(* IEC 61131-3 sources: repolevel_ST_code_completion/output/0122完整版本_无planner目前sota/repoeval_Command1/readful_result_history, 38 files *)

(* ---- FB_AirConComfortCommand_0.st ---- *)
FUNCTION_BLOCK PUBLIC FB_AirConComfortCommand IMPLEMENTS I_Command
VAR
	refAirConditioning : REFERENCE TO FB_AirConditioning;
END_VAR

METHOD Execute : BOOL
VAR
	isValidRef : BOOL;
END_VAR

isValidRef := __ISVALIDREF(refAirConditioning);

IF isValidRef THEN
	refAirConditioning.Activate();
	refAirConditioning.SetTemperature(20.0);
	Execute := TRUE;
ELSE
	Execute := FALSE;
END_IF
END_FUNCTION_BLOCK

(* ---- FB_AirConComfortCommand_1.st ---- *)
FUNCTION_BLOCK PUBLIC FB_AirConComfortCommand IMPLEMENTS I_Command
VAR
  refAirConditioning : REFERENCE TO FB_AirConditioning;
END_VAR

METHOD Execute : BOOL
VAR
  isValidRef : BOOL;
END_VAR

isValidRef := __ISVALIDREF(refAirConditioning);

IF isValidRef THEN
  refAirConditioning.Activate();
  refAirConditioning.SetTemperature(20.0);
  Execute := TRUE;
ELSE
  Execute := FALSE;
END_IF
END_METHOD

(* ---- FB_AirConditioning_0.st ---- *)
FUNCTION_BLOCK PUBLIC FB_AirConditioning
VAR_OUTPUT
	bActive			: BOOL;
	lrTemperature	: LREAL;
END_VAR
VAR
    bInitialized : BOOL := FALSE;
END_VAR

IF NOT bInitialized THEN
    bActive := FALSE;
    lrTemperature := 22.0; // Default temperature
    bInitialized := TRUE;
END_IF;

IF bActive THEN
    // Logic for active air conditioning operation can be added here
ELSE
    // Logic for inactive air conditioning state can be added here
END_IF;
END_FUNCTION_BLOCK

(* ---- FB_AirConditioning_1.st ---- *)
FUNCTION_BLOCK PUBLIC FB_AirConditioning
VAR_OUTPUT
	bActive			: BOOL;
	lrTemperature	: LREAL;
END_VAR
VAR
    bInitialized : BOOL := FALSE;
END_VAR

IF NOT bInitialized THEN
    bActive := FALSE;
    lrTemperature := 22.0; // Default temperature
    bInitialized := TRUE;
END_IF;

IF bActive THEN
    // Logic for active air conditioning operation can be added here
ELSE
    // Logic for inactive air conditioning state can be added here
END_IF;
END_FUNCTION_BLOCK

(* ---- FB_AirConditioning_2.st ---- *)
FUNCTION_BLOCK PUBLIC FB_AirConditioning
VAR_OUTPUT
  bActive			: BOOL;
  lrTemperature	: LREAL;
END_VAR
VAR
  bInitialized : BOOL := FALSE;
END_VAR

IF NOT bInitialized THEN
  bActive := FALSE;
  lrTemperature := 22.0; // Default temperature
  bInitialized := TRUE;
END_IF

IF bActive THEN
  // Logic for active air conditioning operation can be added here
ELSE
  // Logic for inactive air conditioning state can be added here
END_IF
END_FUNCTION_BLOCK

(* ---- FB_AirConditioning_3.st ---- *)
FUNCTION_BLOCK FB_AirConditioning
VAR_OUTPUT
 bActive			: BOOL;
 lrTemperature	: LREAL;
END_VAR
VAR
 bInitialized : BOOL := FALSE;
END_VAR

IF NOT bInitialized THEN
 bActive := FALSE;
 lrTemperature := 22.0; // Default temperature
 bInitialized := TRUE;
END_IF

IF bActive THEN
 // Logic for active air conditioning operation can be added here
ELSE
 // Logic for inactive air conditioning state can be added here
END_IF
END_FUNCTION_BLOCK

(* ---- FB_AirConStandbyCommand_0.st ---- *)
FUNCTION_BLOCK PUBLIC FB_AirConStandbyCommand IMPLEMENTS I_Command
VAR
    refAirConditioning : REFERENCE TO FB_AirConditioning;
END_VAR

IF __ISVALIDREF(refAirConditioning) THEN
    refAirConditioning.bActive := FALSE;
END_IF
END_FUNCTION_BLOCK

(* ---- FB_AirConStandbyCommand_1.st ---- *)
FUNCTION_BLOCK PUBLIC FB_AirConStandbyCommand IMPLEMENTS I_Command
VAR
  refAirConditioning : REFERENCE TO FB_AirConditioning;
END_VAR

IF __ISVALIDREF(refAirConditioning) THEN
  refAirConditioning.bActive := FALSE;
END_IF
// Removed END_FUNCTION_BLOCK as it does not follow Codesys syntax conventions.

(* ---- FB_AirConStandbyCommand_2.st ---- *)
FUNCTION_BLOCK PUBLIC FB_AirConStandbyCommand IMPLEMENTS I_Command
VAR
 refAirConditioning : REFERENCE TO FB_AirConditioning;
END_VAR

IF __ISVALIDREF(refAirConditioning) THEN
 refAirConditioning.bActive := FALSE;
END_IF
// Ensure all operations finalize gracefully. END_FUNCTION_BLOCK keyword avoided as it isn't IEC 61131-3 compliant.

(* ---- FB_AirConStandbyCommand_3.st ---- *)
FUNCTION_BLOCK PUBLIC FB_AirConStandbyCommand IMPLEMENTS I_Command
VAR
refAirConditioning : REFERENCE TO FB_AirConditioning;
END_VAR

IF __ISVALIDREF(refAirConditioning) THEN
refAirConditioning.bActive := FALSE;
END_IF
// Comment removed to maintain clarity and proper IEC 61131-3 formatting.

(* ---- FB_CDPlayer_0.st ---- *)
FUNCTION_BLOCK PUBLIC FB_CDPlayer
VAR_OUTPUT
	bPlayerActive		: BOOL;
	byVolume			: BYTE;
	byTrack				: UINT;
END_VAR
VAR
    bInitialized : BOOL := FALSE;
END_VAR

IF NOT bInitialized THEN
    bPlayerActive := FALSE;
    byVolume := 50; // Default volume level
    byTrack := 1;   // Default track number
    bInitialized := TRUE;
END_IF;

IF bPlayerActive THEN
    // Logic for active player state can be implemented here
END_IF;
END_FUNCTION_BLOCK

(* ---- FB_CDPlayer_1.st ---- *)
FUNCTION_BLOCK PUBLIC FB_CDPlayer
VAR_OUTPUT
	bPlayerActive		: BOOL;
	byVolume			: BYTE;
	byTrack				: UINT;
END_VAR
VAR
    bInitialized : BOOL := FALSE;
END_VAR

IF NOT bInitialized THEN
  bPlayerActive := FALSE;
  byVolume := 50; // Default volume level
  byTrack := 1;   // Default track number
  bInitialized := TRUE;
END_IF

IF bPlayerActive THEN
  // Logic for active player state can be implemented here
END_IF

END_FUNCTION_BLOCK

(* ---- FB_Lamp_0.st ---- *)
FUNCTION_BLOCK PUBLIC FB_Lamp
VAR_OUTPUT
	byLevel			: BYTE;
END_VAR
VAR
    byCurrentLevel : BYTE := 0;
END_VAR

IF byCurrentLevel <> byLevel THEN
    byCurrentLevel := byLevel;
END_IF;
END_FUNCTION_BLOCK

(* ---- FB_Lamp_1.st ---- *)
FUNCTION_BLOCK PUBLIC FB_Lamp
VAR_OUTPUT
  byLevel			: BYTE;
END_VAR
VAR
  byCurrentLevel : BYTE := 0;
END_VAR

IF byCurrentLevel <> byLevel THEN
  byCurrentLevel := byLevel;
END_IF

END_FUNCTION_BLOCK

(* ---- FB_LampSetLevelCommand_0.st ---- *)
FUNCTION_BLOCK PUBLIC FB_LampSetLevelCommand IMPLEMENTS I_Command
VAR
	refLamp		: REFERENCE TO FB_Lamp;
	byNewLevel	: BYTE;
END_VAR

VAR
	isExecuted : BOOL := FALSE;
END_VAR

IF __ISVALIDREF(refLamp) THEN
	refLamp.SetLevel(byNewLevel);
	isExecuted := TRUE;
END_IF
END_FUNCTION_BLOCK

(* ---- FB_LampSetLevelCommand_1.st ---- *)
FUNCTION_BLOCK PUBLIC FB_LampSetLevelCommand IMPLEMENTS I_Command
VAR
  refLamp		: REFERENCE TO FB_Lamp;   // Lamp reference
  byNewLevel	: BYTE;                  // New level to be set
  isExecuted : BOOL := FALSE;          // Execution status
END_VAR

IF __ISVALIDREF(refLamp) THEN
  refLamp.SetLevel(byNewLevel);        // Set the lamp level
  isExecuted := TRUE;                 // Mark command as executed
END_IF
END_FUNCTION_BLOCK

(* ---- FB_MusicPlayCommand_0.st ---- *)
FUNCTION_BLOCK PUBLIC FB_MusicPlayCommand IMPLEMENTS I_Command
VAR
	refCDPlayer : REFERENCE TO FB_CDPlayer;
END_VAR

METHOD Execute
VAR
	refCDPlayer : REFERENCE TO FB_CDPlayer;
END_VAR

IF (__ISVALIDREF(THIS^.refCDPlayer)) THEN
	THIS^.refCDPlayer.SetVolume(40);
	THIS^.refCDPlayer.SetTrack(1);
	THIS^.refCDPlayer.Start();
END_IF
END_FUNCTION_BLOCK

(* ---- FB_MusicPlayCommand_1.st ---- *)
FUNCTION_BLOCK PUBLIC FB_MusicPlayCommand IMPLEMENTS I_Command
VAR
	refCDPlayer : REFERENCE TO FB_CDPlayer;
END_VAR

METHOD Execute

IF (__ISVALIDREF(THIS^.refCDPlayer)) THEN
  THIS^.refCDPlayer.SetVolume(40);
  THIS^.refCDPlayer.SetTrack(1);
  THIS^.refCDPlayer.Start();
END_IF
END_FUNCTION_BLOCK

(* ---- FB_MusicPlayCommand_2.st ---- *)
FUNCTION_BLOCK PUBLIC FB_MusicPlayCommand IMPLEMENTS I_Command
VAR
	refCDPlayer : REFERENCE TO FB_CDPlayer;
END_VAR

METHOD Execute

IF (__ISVALIDREF(THIS^.refCDPlayer)) THEN
 // Ensure all referenced methods are valid and accessible.
 THIS^.refCDPlayer.SetVolume(40); // Example: Volume level
 THIS^.refCDPlayer.SetTrack(1);   // Example: Track number
 THIS^.refCDPlayer.Start();       // Begin playback
END_IF
END_FUNCTION_BLOCK

(* ---- FB_MusicPlayCommand_3.st ---- *)
FUNCTION_BLOCK PUBLIC FB_MusicPlayCommand IMPLEMENTS I_Command
VAR
	refCDPlayer : REFERENCE TO FB_CDPlayer;
END_VAR

METHOD Execute

IF (__ISVALIDREF(THIS^.refCDPlayer)) THEN
// Ensure all referenced methods are valid and accessible.
THIS^.refCDPlayer.SetVolume(40); // Example: Volume level
THIS^.refCDPlayer.SetTrack(1);   // Example: Track number
THIS^.refCDPlayer.Start();       // Begin playback
ELSE
// Handle the invalid reference case by adding a comment or logging here, if necessary.
// Since new variables cannot be declared, no additional action is taken here.
END_IF
END_FUNCTION_BLOCK

(* ---- FB_MusicStopCommand_0.st ---- *)
FUNCTION_BLOCK PUBLIC FB_MusicStopCommand IMPLEMENTS I_Command
VAR
	refCDPlayer : REFERENCE TO FB_CDPlayer;
END_VAR

METHOD Execute
VAR
	refCDPlayer : REFERENCE TO FB_CDPlayer;
END_VAR

IF (__ISVALIDREF(THIS^.refCDPlayer)) THEN
	THIS^.refCDPlayer.Stop();
END_IF
END_FUNCTION_BLOCK

(* ---- FB_MusicStopCommand_1.st ---- *)
FUNCTION_BLOCK PUBLIC FB_MusicStopCommand IMPLEMENTS I_Command
VAR
	refCDPlayer : REFERENCE TO FB_CDPlayer;
END_VAR

METHOD Execute

IF (__ISVALIDREF(THIS^.refCDPlayer)) THEN
  THIS^.refCDPlayer.Stop();
END_IF
END_FUNCTION_BLOCK

(* ---- FB_MusicStopCommand_2.st ---- *)
FUNCTION_BLOCK PUBLIC FB_MusicStopCommand IMPLEMENTS I_Command
VAR
	refCDPlayer : REFERENCE TO FB_CDPlayer;
END_VAR

METHOD Execute

IF (__ISVALIDREF(THIS^.refCDPlayer)) THEN
 IF THIS^.refCDPlayer <> 0 THEN // Ensure refCDPlayer is assigned
  THIS^.refCDPlayer.Stop();
 END_IF;
END_IF
END_FUNCTION_BLOCK

(* ---- FB_MusicStopCommand_3.st ---- *)
FUNCTION_BLOCK PUBLIC FB_MusicStopCommand IMPLEMENTS I_Command
VAR
	refCDPlayer : REFERENCE TO FB_CDPlayer;
END_VAR

METHOD Execute

IF (__ISVALIDREF(THIS^.refCDPlayer)) THEN
 THIS^.refCDPlayer.Stop();
END_IF
END_FUNCTION_BLOCK

(* ---- FB_Socket_0.st ---- *)
FUNCTION_BLOCK PUBLIC FB_Socket
VAR_OUTPUT
	bActive		: BOOL;
END_VAR
VAR
    bInitialized : BOOL := FALSE;
END_VAR

IF NOT bInitialized THEN
    bActive := FALSE;
    bInitialized := TRUE;
END_IF;
END_FUNCTION_BLOCK

(* ---- FB_Socket_1.st ---- *)
FUNCTION_BLOCK PUBLIC FB_Socket
VAR_OUTPUT
	bActive		: BOOL;
END_VAR
VAR
    bInitialized : BOOL := FALSE;
END_VAR

IF NOT bInitialized THEN
    bActive := FALSE;
    bInitialized := TRUE;
END_IF;
END_FUNCTION_BLOCK

(* ---- FB_SocketOffCommand_0.st ---- *)
FUNCTION_BLOCK PUBLIC FB_SocketOffCommand IMPLEMENTS I_Command
VAR
    refSocket : REFERENCE TO FB_Socket;
END_VAR

VAR
    bIsValidRef : BOOL;
END_VAR

bIsValidRef := __ISVALIDREF(refSocket);

IF bIsValidRef THEN
    refSocket.Off();
END_IF
END_FUNCTION_BLOCK

(* ---- FB_SocketOffCommand_1.st ---- *)
FUNCTION_BLOCK PUBLIC FB_SocketOffCommand IMPLEMENTS I_Command
VAR
  refSocket : REFERENCE TO FB_Socket;
END_VAR

VAR
  bIsValidRef : BOOL;
END_VAR

// Check if the reference is valid
IF __ISVALIDREF(refSocket) THEN
  bIsValidRef := TRUE;
  refSocket.Off(); // Call the Off method of the referenced instance
ELSE
  bIsValidRef := FALSE; // The reference is invalid
END_IF

END_FUNCTION_BLOCK

(* ---- FB_SocketOffCommand_2.st ---- *)
FUNCTION_BLOCK PUBLIC FB_SocketOffCommand IMPLEMENTS I_Command
VAR
 refSocket : REFERENCE TO FB_Socket;
END_VAR

VAR
 bIsValidRef : BOOL;
END_VAR

// Check if the reference is valid
bIsValidRef := __ISVALIDREF(refSocket); // Update bIsValidRef based on reference validity

IF bIsValidRef THEN
 refSocket.Off(); // Call the Off method of the referenced instance if valid
END_IF

END_FUNCTION_BLOCK

(* ---- FB_SocketOffCommand_3.st ---- *)
FUNCTION_BLOCK PUBLIC FB_SocketOffCommand IMPLEMENTS I_Command
VAR
refSocket : REFERENCE TO FB_Socket;
END_VAR

VAR
bIsValidRef : BOOL;
END_VAR

// Check if the reference is valid
IF __ISVALIDREF(refSocket) THEN
refSocket.Off(); // Call the Off method of the referenced instance if valid
bIsValidRef := TRUE; // Set bIsValidRef to TRUE
ELSE
bIsValidRef := FALSE; // Set bIsValidRef to FALSE if reference is invalid
END_IF

END_FUNCTION_BLOCK

(* ---- FB_SocketOnCommand_0.st ---- *)
FUNCTION_BLOCK PUBLIC FB_SocketOnCommand IMPLEMENTS I_Command
VAR
	refSocket : REFERENCE TO FB_Socket;
END_VAR

METHOD Execute : BOOL
VAR
	isExecuted : BOOL := FALSE;
END_VAR

IF __ISVALIDREF(refSocket) THEN
	refSocket.On();
	isExecuted := TRUE;
END_IF

Execute := isExecuted;
END_FUNCTION_BLOCK

(* ---- FB_SocketOnCommand_1.st ---- *)
FUNCTION_BLOCK PUBLIC FB_SocketOnCommand IMPLEMENTS I_Command
VAR
	refSocket : REFERENCE TO FB_Socket;
END_VAR

METHOD Execute : BOOL
VAR
	isExecuted : BOOL := FALSE;
END_VAR

IF __ISVALIDREF(refSocket) THEN
	refSocket.On();
	isExecuted := TRUE;
END_IF

RETURN;
END_FUNCTION_BLOCK

(* ---- FB_SocketOnCommand_2.st ---- *)
FUNCTION_BLOCK PUBLIC FB_SocketOnCommand IMPLEMENTS I_Command
VAR
	refSocket : REFERENCE TO FB_Socket;
END_VAR

METHOD Execute : BOOL
IF __ISVALIDREF(refSocket) THEN
  refSocket.On();
  Execute := TRUE; // Assign return value directly
ELSE
  Execute := FALSE; // Default case for return value
END_IF

RETURN;
END_FUNCTION_BLOCK

(* ---- FB_SocketOnCommand_3.st ---- *)
FUNCTION_BLOCK PUBLIC FB_SocketOnCommand IMPLEMENTS I_Command
VAR
	refSocket : REFERENCE TO FB_Socket;
END_VAR

METHOD Execute : BOOL
IF __ISVALIDREF(refSocket) THEN
 refSocket.On();
 Execute := TRUE; // Last value of Execute is managed here
ELSE
 Execute := FALSE; // Default case for Execute
END_IF
END_METHOD // No explicit RETURN needed for METHOD
END_FUNCTION_BLOCK

(* ---- FB_SwitchPanel_0.st ---- *)
FUNCTION_BLOCK PUBLIC FB_SwitchPanel
VAR_INPUT
	arrSwitch		: ARRAY[1..8] OF BOOL;
END_VAR
VAR
	aiCommand		: ARRAY[1..8] OF I_Command;
	arrRtrig		: ARRAY[1..8] OF R_TRIG;
	nIndex			: INT;
END_VAR

FOR nIndex := 1 TO 8 DO
	arrRtrig[nIndex](CLK := arrSwitch[nIndex]);
	IF arrRtrig[nIndex].Q THEN
		IF (aiCommand[nIndex] <> 0) THEN
			aiCommand[nIndex].Execute();
		END_IF
	END_IF
END_FOR
END_FUNCTION_BLOCK

(* ---- FB_SwitchPanel_1.st ---- *)
FUNCTION_BLOCK PUBLIC FB_SwitchPanel
VAR_INPUT
	arrSwitch		: ARRAY[1..8] OF BOOL;
END_VAR
VAR
	aiCommand		: ARRAY[1..8] OF I_Command;
	arrRtrig		: ARRAY[1..8] OF R_TRIG;
	nIndex			: INT;
END_VAR

FOR nIndex := 1 TO 8 DO
  arrRtrig[nIndex](CLK := arrSwitch[nIndex]); // Trigger rising edge detection
  IF arrRtrig[nIndex].Q THEN
    IF aiCommand[nIndex].Valid THEN // Check for a valid I_Command instance
      aiCommand[nIndex](Execute := TRUE); // Correctly invoke the Execute input of the function block
    END_IF
  END_IF
END_FOR
END_FUNCTION_BLOCK

(* ---- FB_SwitchPanel_2.st ---- *)
FUNCTION_BLOCK PUBLIC FB_SwitchPanel
VAR_INPUT
	arrSwitch		: ARRAY[1..8] OF BOOL;
END_VAR
VAR
	aiCommand		: ARRAY[1..8] OF I_Command;
	arrRtrig		: ARRAY[1..8] OF R_TRIG;
	nIndex			: INT;
END_VAR

FOR nIndex := 1 TO 8 DO
 arrRtrig[nIndex](CLK := arrSwitch[nIndex]); // Trigger rising edge detection
 IF arrRtrig[nIndex].Q THEN
  aiCommand[nIndex](Execute := TRUE); // Invoke the Execute input of the function block directly
 END_IF
END_FOR
END_FUNCTION_BLOCK

(* ---- FB_SwitchPanel_3.st ---- *)
FUNCTION_BLOCK PUBLIC FB_SwitchPanel
VAR_INPUT
	arrSwitch		: ARRAY[1..8] OF BOOL;
END_VAR
VAR
	aiCommand		: ARRAY[1..8] OF I_Command;
	arrRtrig		: ARRAY[1..8] OF R_TRIG;
	nIndex			: INT;
END_VAR

FOR nIndex := 1 TO 8 DO
arrRtrig[nIndex](CLK := arrSwitch[nIndex]); // Trigger rising edge detection
IF arrRtrig[nIndex].Q THEN
 IF aiCommand[nIndex].Execute <> 0 THEN // Ensure the function block instance is valid
 aiCommand[nIndex](Execute := TRUE); // Invoke the Execute input of the function block
 END_IF
END_IF
END_FOR
END_FUNCTION_BLOCK
